// TIA Portal V18 export
TYPE "LGasp_type_lubrificazioniPC"
// stored: IsFailsafeCompliant false
   STRUCT
      tipo : Int;   // DA DEFINIRE
      nome : WString;   // nome lubrificazione visualizzato nel PC
      nometrad : WString;   // nome lubrificazione visualizzato nel PC seconda lingua
      cmdabilitata : Bool;   // segnale toggle da PC, abilitata in automatico
      cmdmanuale : Bool;   // segnaleda PC, comando lubrificazione
      cmddurata : LReal;   // durata lubrificazione
      cmdquota : LReal;   // quota abilitazione lubrificazione
      stsquotaattuale : LReal;   // quota attualmente fatta
      cmdnumcolpi : LReal;   // numero colpi attivazione lubrificazione
      stsnumcolpiattuali : LReal;   // numero colpi attualmente fatti
      cmdritardo : LReal;   // ritardo attivazione lubrificazione
      stsRitardoattuale : LReal;   // ritardo stato attuale
   END_STRUCT;
END_TYPE
